    movel([0.091706, -1.408283, -2.552666, -0.751440, 1.570796, 1.662503],accel_mss,speed_ms,0,blend_radius_m)
    movel([0.089171, -1.432149, -2.534440, -0.745800, 1.570796, 1.659968],accel_mss,speed_ms,0,blend_radius_m)
    movel([0.086775, -1.455223, -2.515999, -0.741166, 1.570796, 1.657571],accel_mss,speed_ms,0,blend_radius_m)
    movel([0.116068, -1.448017, -2.521846, -0.742526, 1.570796, 1.686864],accel_mss,speed_ms,0,blend_radius_m)
    movel([0.118372, -1.447476, -2.522281, -0.742631, 1.570796, 1.689168],accel_mss,speed_ms,0,blend_radius_m)
    speed_ms = 0.005
    movel([0.118372, -1.439256, -2.518569, -0.754564, 1.570796, 1.689168],accel_mss,speed_ms,0,blend_radius_m)
    speed_ms = 0.040
    movel([0.108373, -1.430908, -2.525151, -0.756330, 1.570796, 1.679169],accel_mss,speed_ms,0,blend_radius_m)
    speed_ms = 0.005
    movel([0.108373, -1.439191, -2.528898, -0.744300, 1.570796, 1.679169],accel_mss,speed_ms,0,blend_radius_m)
    speed_ms = 0.030
    movel([0.109064, -1.438479, -2.529462, -0.744448, 1.570796, 1.679861],accel_mss,speed_ms,0,blend_radius_m)
    movel([0.109634, -1.437741, -2.530045, -0.744603, 1.570796, 1.680430],accel_mss,speed_ms,0,blend_radius_m)
    movel([0.110059, -1.437005, -2.530627, -0.744758, 1.570796, 1.680855],accel_mss,speed_ms,0,blend_radius_m)
    movel([0.110328, -1.436288, -2.531192, -0.744909, 1.570796, 1.681124],accel_mss,speed_ms,0,blend_radius_m)
    movel([0.110489, -1.435357, -2.531925, -0.745107, 1.570796, 1.681285],accel_mss,speed_ms,0,blend_radius_m)
    movel([0.110459, -1.434480, -2.532614, -0.745295, 1.570796, 1.681255],accel_mss,speed_ms,0,blend_radius_m)
    movel([0.110228, -1.433791, -2.533154, -0.745444, 1.570796, 1.681024],accel_mss,speed_ms,0,blend_radius_m)
    movel([0.109775, -1.433248, -2.533580, -0.745561, 1.570796, 1.680572],accel_mss,speed_ms,0,blend_radius_m)
    movel([0.109099, -1.432863, -2.533881, -0.745645, 1.570796, 1.679896],accel_mss,speed_ms,0,blend_radius_m)
    movel([0.108266, -1.432676, -2.534028, -0.745685, 1.570796, 1.679062],accel_mss,speed_ms,0,blend_radius_m)
    movel([0.107167, -1.432651, -2.534047, -0.745691, 1.570796, 1.677964],accel_mss,speed_ms,0,blend_radius_m)
    movel([0.106011, -1.432776, -2.533950, -0.745663, 1.570796, 1.676807],accel_mss,speed_ms,0,blend_radius_m)
    movel([0.104600, -1.433064, -2.533724, -0.745601, 1.570796, 1.675397],accel_mss,speed_ms,0,blend_radius_m)
    movel([0.103766, -1.433387, -2.533471, -0.745531, 1.570796, 1.674563],accel_mss,speed_ms,0,blend_radius_m)
    movel([0.103005, -1.433924, -2.533050, -0.745415, 1.570796, 1.673801],accel_mss,speed_ms,0,blend_radius_m)
    movel([0.101867, -1.435005, -2.532202, -0.745183, 1.570796, 1.672664],accel_mss,speed_ms,0,blend_radius_m)
    movel([0.100937, -1.436006, -2.531414, -0.744969, 1.570796, 1.671733],accel_mss,speed_ms,0,blend_radius_m)
    movel([0.100376, -1.436776, -2.530807, -0.744806, 1.570796, 1.671172],accel_mss,speed_ms,0,blend_radius_m)
    movel([0.100054, -1.437509, -2.530228, -0.744651, 1.570796, 1.670850],accel_mss,speed_ms,0,blend_radius_m)
    movel([0.099878, -1.438369, -2.529549, -0.744471, 1.570796, 1.670674],accel_mss,speed_ms,0,blend_radius_m)
    movel([0.099866, -1.438969, -2.529074, -0.744346, 1.570796, 1.670663],accel_mss,speed_ms,0,blend_radius_m)
    movel([0.099966, -1.439526, -2.528633, -0.744230, 1.570796, 1.670762],accel_mss,speed_ms,0,blend_radius_m)
    movel([0.100487, -1.440458, -2.527893, -0.744038, 1.570796, 1.671284],accel_mss,speed_ms,0,blend_radius_m)
    movel([0.100905, -1.440826, -2.527601, -0.743962, 1.570796, 1.671701],accel_mss,speed_ms,0,blend_radius_m)
    movel([0.101980, -1.441312, -2.527214, -0.743863, 1.570796, 1.672776],accel_mss,speed_ms,0,blend_radius_m)
    movel([0.102614, -1.441422, -2.527127, -0.743840, 1.570796, 1.673411],accel_mss,speed_ms,0,blend_radius_m)
    movel([0.104044, -1.441369, -2.527169, -0.743851, 1.570796, 1.674840],accel_mss,speed_ms,0,blend_radius_m)
    movel([0.104799, -1.441206, -2.527298, -0.743884, 1.570796, 1.675596],accel_mss,speed_ms,0,blend_radius_m)
    movel([0.106310, -1.440622, -2.527762, -0.744004, 1.570796, 1.677107],accel_mss,speed_ms,0,blend_radius_m)
    movel([0.107038, -1.440213, -2.528087, -0.744088, 1.570796, 1.677835],accel_mss,speed_ms,0,blend_radius_m)
    movel([0.108373, -1.439191, -2.528898, -0.744300, 1.570796, 1.679169],accel_mss,speed_ms,0,blend_radius_m)
    movel([0.109064, -1.438479, -2.529462, -0.744448, 1.570796, 1.679861],accel_mss,speed_ms,0,blend_radius_m)
    movel([0.109634, -1.437741, -2.530045, -0.744603, 1.570796, 1.680430],accel_mss,speed_ms,0,blend_radius_m)
    movel([0.109919, -1.437246, -2.530436, -0.744707, 1.570796, 1.680715],accel_mss,speed_ms,0,blend_radius_m)
    speed_ms = 0.005
    movel([0.109919, -1.428948, -2.526681, -0.756760, 1.570796, 1.680715],accel_mss,speed_ms,0,blend_radius_m)
    speed_ms = 0.040
    movel([0.118670, -1.416855, -2.535995, -0.759539, 1.570796, 1.689466],accel_mss,speed_ms,0,blend_radius_m)
    speed_ms = 0.005
    movel([0.118670, -1.425243, -2.539801, -0.747344, 1.570796, 1.689466],accel_mss,speed_ms,0,blend_radius_m)
    speed_ms = 0.030
    movel([0.124083, -1.423937, -2.540808, -0.747644, 1.570796, 1.694879],accel_mss,speed_ms,0,blend_radius_m)
    movel([0.117797, -1.434992, -2.532211, -0.745185, 1.570796, 1.688593],accel_mss,speed_ms,0,blend_radius_m)
    movel([0.117485, -1.435414, -2.531880, -0.745095, 1.570796, 1.688282],accel_mss,speed_ms,0,blend_radius_m)
    movel([0.116691, -1.434317, -2.532742, -0.745330, 1.570796, 1.687488],accel_mss,speed_ms,0,blend_radius_m)
    movel([0.115225, -1.431178, -2.535198, -0.746013, 1.570796, 1.686021],accel_mss,speed_ms,0,blend_radius_m)
    movel([0.113262, -1.426570, -2.538777, -0.747042, 1.570796, 1.684058],accel_mss,speed_ms,0,blend_radius_m)
    movel([0.118670, -1.425243, -2.539801, -0.747344, 1.570796, 1.689466],accel_mss,speed_ms,0,blend_radius_m)
    movel([0.121038, -1.424669, -2.540244, -0.747476, 1.570796, 1.691834],accel_mss,speed_ms,0,blend_radius_m)
    speed_ms = 0.005
    movel([0.121038, -1.416276, -2.536436, -0.759677, 1.570796, 1.691834],accel_mss,speed_ms,0,blend_radius_m)
    speed_ms = 0.040
    movel([0.111498, -1.424285, -2.530298, -0.757806, 1.570796, 1.682294],accel_mss,speed_ms,0,blend_radius_m)
    speed_ms = 0.005
    movel([0.111498, -1.432618, -2.534073, -0.745698, 1.570796, 1.682294],accel_mss,speed_ms,0,blend_radius_m)
    speed_ms = 0.030
    movel([0.111769, -1.433135, -2.533668, -0.745586, 1.570796, 1.682566],accel_mss,speed_ms,0,blend_radius_m)
    movel([0.112066, -1.434546, -2.532562, -0.745281, 1.570796, 1.682862],accel_mss,speed_ms,0,blend_radius_m)
    movel([0.112043, -1.435207, -2.532042, -0.745139, 1.570796, 1.682839],accel_mss,speed_ms,0,blend_radius_m)
    movel([0.111849, -1.436112, -2.531330, -0.744947, 1.570796, 1.682646],accel_mss,speed_ms,0,blend_radius_m)
    movel([0.111503, -1.437034, -2.530604, -0.744751, 1.570796, 1.682299],accel_mss,speed_ms,0,blend_radius_m)
    movel([0.111013, -1.437950, -2.529880, -0.744559, 1.570796, 1.681809],accel_mss,speed_ms,0,blend_radius_m)
    movel([0.110389, -1.438840, -2.529176, -0.744373, 1.570796, 1.681185],accel_mss,speed_ms,0,blend_radius_m)
    movel([0.109649, -1.439681, -2.528510, -0.744198, 1.570796, 1.680445],accel_mss,speed_ms,0,blend_radius_m)
    movel([0.108810, -1.440452, -2.527898, -0.744039, 1.570796, 1.679607],accel_mss,speed_ms,0,blend_radius_m)
    movel([0.107889, -1.441141, -2.527350, -0.743898, 1.570796, 1.678685],accel_mss,speed_ms,0,blend_radius_m)
    movel([0.106909, -1.441727, -2.526884, -0.743778, 1.570796, 1.677706],accel_mss,speed_ms,0,blend_radius_m)
    movel([0.105881, -1.442207, -2.526502, -0.743680, 1.570796, 1.676677],accel_mss,speed_ms,0,blend_radius_m)
    movel([0.104840, -1.442562, -2.526218, -0.743608, 1.570796, 1.675636],accel_mss,speed_ms,0,blend_radius_m)
    movel([0.103811, -1.442784, -2.526041, -0.743563, 1.570796, 1.674607],accel_mss,speed_ms,0,blend_radius_m)
    movel([0.102814, -1.442870, -2.525973, -0.743546, 1.570796, 1.673610],accel_mss,speed_ms,0,blend_radius_m)
    movel([0.101860, -1.442821, -2.526012, -0.743556, 1.570796, 1.672657],accel_mss,speed_ms,0,blend_radius_m)
    movel([0.100981, -1.442635, -2.526161, -0.743594, 1.570796, 1.671777],accel_mss,speed_ms,0,blend_radius_m)
    movel([0.100198, -1.442319, -2.526412, -0.743658, 1.570796, 1.670994],accel_mss,speed_ms,0,blend_radius_m)
    movel([0.099523, -1.441881, -2.526762, -0.743747, 1.570796, 1.670319],accel_mss,speed_ms,0,blend_radius_m)
    movel([0.098634, -1.440907, -2.527537, -0.743946, 1.570796, 1.669430],accel_mss,speed_ms,0,blend_radius_m)
    movel([0.098355, -1.440381, -2.527954, -0.744054, 1.570796, 1.669152],accel_mss,speed_ms,0,blend_radius_m)
    movel([0.098129, -1.439183, -2.528904, -0.744301, 1.570796, 1.668926],accel_mss,speed_ms,0,blend_radius_m)
    movel([0.098186, -1.438537, -2.529416, -0.744436, 1.570796, 1.668982],accel_mss,speed_ms,0,blend_radius_m)
    movel([0.098626, -1.437145, -2.530516, -0.744728, 1.570796, 1.669422],accel_mss,speed_ms,0,blend_radius_m)
    movel([0.099087, -1.436285, -2.531194, -0.744910, 1.570796, 1.669883],accel_mss,speed_ms,0,blend_radius_m)
    movel([0.099671, -1.435447, -2.531853, -0.745088, 1.570796, 1.670467],accel_mss,speed_ms,0,blend_radius_m)
    movel([0.100365, -1.434653, -2.532478, -0.745258, 1.570796, 1.671161],accel_mss,speed_ms,0,blend_radius_m)
    movel([0.101155, -1.433915, -2.533057, -0.745417, 1.570796, 1.671952],accel_mss,speed_ms,0,blend_radius_m)
    movel([0.102056, -1.433221, -2.533601, -0.745567, 1.570796, 1.672852],accel_mss,speed_ms,0,blend_radius_m)
    movel([0.103011, -1.432609, -2.534081, -0.745700, 1.570796, 1.673808],accel_mss,speed_ms,0,blend_radius_m)
    movel([0.104006, -1.432092, -2.534485, -0.745813, 1.570796, 1.674803],accel_mss,speed_ms,0,blend_radius_m)
    movel([0.105024, -1.431675, -2.534810, -0.745904, 1.570796, 1.675820],accel_mss,speed_ms,0,blend_radius_m)
    movel([0.106037, -1.431373, -2.535046, -0.745970, 1.570796, 1.676834],accel_mss,speed_ms,0,blend_radius_m)
    movel([0.107034, -1.431190, -2.535189, -0.746010, 1.570796, 1.677830],accel_mss,speed_ms,0,blend_radius_m)
    movel([0.108000, -1.431125, -2.535240, -0.746025, 1.570796, 1.678796],accel_mss,speed_ms,0,blend_radius_m)
    movel([0.108911, -1.431181, -2.535196, -0.746012, 1.570796, 1.679707],accel_mss,speed_ms,0,blend_radius_m)
    movel([0.109713, -1.431357, -2.535058, -0.745973, 1.570796, 1.680510],accel_mss,speed_ms,0,blend_radius_m)
    movel([0.110423, -1.431660, -2.534822, -0.745907, 1.570796, 1.681220],accel_mss,speed_ms,0,blend_radius_m)
    movel([0.111022, -1.432085, -2.534490, -0.745814, 1.570796, 1.681818],accel_mss,speed_ms,0,blend_radius_m)
    movel([0.111498, -1.432618, -2.534073, -0.745698, 1.570796, 1.682294],accel_mss,speed_ms,0,blend_radius_m)
    movel([0.111769, -1.433135, -2.533668, -0.745586, 1.570796, 1.682566],accel_mss,speed_ms,0,blend_radius_m)
    movel([0.112020, -1.434323, -2.532737, -0.745329, 1.570796, 1.682816],accel_mss,speed_ms,0,blend_radius_m)
    speed_ms = 0.005
    movel([0.112020, -1.426003, -2.528969, -0.757417, 1.570796, 1.682816],accel_mss,speed_ms,0,blend_radius_m)
    speed_ms = 0.040
    movel([0.108450, -1.426614, -2.528496, -0.757279, 1.570796, 1.679246],accel_mss,speed_ms,0,blend_radius_m)
    speed_ms = 0.005
    movel([0.108450, -1.434929, -2.532261, -0.745199, 1.570796, 1.679246],accel_mss,speed_ms,0,blend_radius_m)
    speed_ms = 0.030
    movel([0.107952, -1.434276, -2.532774, -0.745339, 1.570796, 1.678748],accel_mss,speed_ms,0,blend_radius_m)
    movel([0.107572, -1.434065, -2.532940, -0.745384, 1.570796, 1.678368],accel_mss,speed_ms,0,blend_radius_m)
    movel([0.107121, -1.433941, -2.533037, -0.745411, 1.570796, 1.677918],accel_mss,speed_ms,0,blend_radius_m)
    movel([0.106038, -1.433948, -2.533031, -0.745410, 1.570796, 1.676835],accel_mss,speed_ms,0,blend_radius_m)
    movel([0.104871, -1.434291, -2.532762, -0.745336, 1.570796, 1.675667],accel_mss,speed_ms,0,blend_radius_m)
    movel([0.103728, -1.434938, -2.532254, -0.745197, 1.570796, 1.674524],accel_mss,speed_ms,0,blend_radius_m)
    movel([0.102745, -1.435815, -2.531564, -0.745010, 1.570796, 1.673541],accel_mss,speed_ms,0,blend_radius_m)
    movel([0.102363, -1.436294, -2.531187, -0.744908, 1.570796, 1.673159],accel_mss,speed_ms,0,blend_radius_m)
    movel([0.101858, -1.437301, -2.530393, -0.744695, 1.570796, 1.672655],accel_mss,speed_ms,0,blend_radius_m)
    movel([0.101749, -1.437800, -2.529999, -0.744590, 1.570796, 1.672545],accel_mss,speed_ms,0,blend_radius_m)
    movel([0.101790, -1.438633, -2.529340, -0.744416, 1.570796, 1.672586],accel_mss,speed_ms,0,blend_radius_m)
    movel([0.102119, -1.439326, -2.528791, -0.744272, 1.570796, 1.672915],accel_mss,speed_ms,0,blend_radius_m)
    movel([0.102703, -1.439804, -2.528412, -0.744173, 1.570796, 1.673500],accel_mss,speed_ms,0,blend_radius_m)
    movel([0.103505, -1.440030, -2.528233, -0.744126, 1.570796, 1.674302],accel_mss,speed_ms,0,blend_radius_m)
    movel([0.104454, -1.439989, -2.528265, -0.744135, 1.570796, 1.675251],accel_mss,speed_ms,0,blend_radius_m)
    movel([0.105461, -1.439681, -2.528509, -0.744198, 1.570796, 1.676258],accel_mss,speed_ms,0,blend_radius_m)
    movel([0.106463, -1.439130, -2.528947, -0.744313, 1.570796, 1.677259],accel_mss,speed_ms,0,blend_radius_m)
    movel([0.107355, -1.438395, -2.529529, -0.744466, 1.570796, 1.678151],accel_mss,speed_ms,0,blend_radius_m)
    movel([0.108163, -1.437463, -2.530265, -0.744661, 1.570796, 1.678959],accel_mss,speed_ms,0,blend_radius_m)
    movel([0.108589, -1.436654, -2.530904, -0.744832, 1.570796, 1.679385],accel_mss,speed_ms,0,blend_radius_m)
    movel([0.108678, -1.435849, -2.531537, -0.745002, 1.570796, 1.679474],accel_mss,speed_ms,0,blend_radius_m)
    movel([0.108450, -1.434929, -2.532261, -0.745199, 1.570796, 1.679246],accel_mss,speed_ms,0,blend_radius_m)
    movel([0.107952, -1.434276, -2.532774, -0.745339, 1.570796, 1.678748],accel_mss,speed_ms,0,blend_radius_m)
    movel([0.107572, -1.434065, -2.532940, -0.745384, 1.570796, 1.678368],accel_mss,speed_ms,0,blend_radius_m)
    movel([0.107121, -1.433941, -2.533037, -0.745411, 1.570796, 1.677918],accel_mss,speed_ms,0,blend_radius_m)
    speed_ms = 0.005
    movel([0.107012, -1.425618, -2.529268, -0.757504, 1.570796, 1.677809],accel_mss,speed_ms,0,blend_radius_m)
    speed_ms = 0.040
    movel([0.083343, -1.436462, -2.520784, -0.755143, 1.570796, 1.654139],accel_mss,speed_ms,0,blend_radius_m)
    speed_ms = 0.005
    movel([0.083343, -1.444703, -2.524508, -0.743178, 1.570796, 1.654139],accel_mss,speed_ms,0,blend_radius_m)
    speed_ms = 0.030
    movel([0.085200, -1.444214, -2.524899, -0.743276, 1.570796, 1.655996],accel_mss,speed_ms,0,blend_radius_m)
    movel([0.085840, -1.437885, -2.529932, -0.744572, 1.570796, 1.656636],accel_mss,speed_ms,0,blend_radius_m)
    movel([0.086489, -1.431498, -2.534949, -0.745943, 1.570796, 1.657285],accel_mss,speed_ms,0,blend_radius_m)
    movel([0.084603, -1.432003, -2.534554, -0.745832, 1.570796, 1.655399],accel_mss,speed_ms,0,blend_radius_m)
    movel([0.082718, -1.432510, -2.534157, -0.745721, 1.570796, 1.653514],accel_mss,speed_ms,0,blend_radius_m)
    movel([0.082098, -1.438881, -2.529144, -0.744364, 1.570796, 1.652894],accel_mss,speed_ms,0,blend_radius_m)
    movel([0.081487, -1.445194, -2.524114, -0.743080, 1.570796, 1.652283],accel_mss,speed_ms,0,blend_radius_m)
    movel([0.083343, -1.444703, -2.524508, -0.743178, 1.570796, 1.654139],accel_mss,speed_ms,0,blend_radius_m)
    movel([0.085200, -1.444214, -2.524899, -0.743276, 1.570796, 1.655996],accel_mss,speed_ms,0,blend_radius_m)
    movel([0.085240, -1.443820, -2.525214, -0.743355, 1.570796, 1.656036],accel_mss,speed_ms,0,blend_radius_m)
    speed_ms = 0.005
    movel([0.085240, -1.435572, -2.521486, -0.755330, 1.570796, 1.656036],accel_mss,speed_ms,0,blend_radius_m)
    speed_ms = 0.040
    movel([0.080369, -1.396684, -2.551051, -0.764654, 1.570796, 1.651165],accel_mss,speed_ms,0,blend_radius_m)
    speed_ms = 0.005
    movel([0.080369, -1.405221, -2.554943, -0.752225, 1.570796, 1.651165],accel_mss,speed_ms,0,blend_radius_m)
    speed_ms = 0.030
    movel([0.082668, -1.404286, -2.555636, -0.752468, 1.570796, 1.653464],accel_mss,speed_ms,0,blend_radius_m)
    movel([0.083132, -1.399509, -2.559154, -0.753727, 1.570796, 1.653929],accel_mss,speed_ms,0,blend_radius_m)
    movel([0.083285, -1.397676, -2.560495, -0.754219, 1.570796, 1.654081],accel_mss,speed_ms,0,blend_radius_m)
    movel([0.083369, -1.394878, -2.562532, -0.754979, 1.570796, 1.654165],accel_mss,speed_ms,0,blend_radius_m)
    movel([0.071293, -1.397205, -2.560838, -0.754346, 1.570796, 1.642090],accel_mss,speed_ms,0,blend_radius_m)
    movel([0.066805, -1.398147, -2.560151, -0.754092, 1.570796, 1.637601],accel_mss,speed_ms,0,blend_radius_m)
    movel([0.059543, -1.399830, -2.558918, -0.753641, 1.570796, 1.630340],accel_mss,speed_ms,0,blend_radius_m)
    movel([0.058947, -1.400083, -2.558732, -0.753573, 1.570796, 1.629743],accel_mss,speed_ms,0,blend_radius_m)
    movel([0.058527, -1.400449, -2.558464, -0.753476, 1.570796, 1.629324],accel_mss,speed_ms,0,blend_radius_m)
    movel([0.058288, -1.400892, -2.558139, -0.753359, 1.570796, 1.629084],accel_mss,speed_ms,0,blend_radius_m)
    movel([0.058040, -1.402395, -2.557032, -0.752962, 1.570796, 1.628837],accel_mss,speed_ms,0,blend_radius_m)
    movel([0.058173, -1.404016, -2.555835, -0.752538, 1.570796, 1.628969],accel_mss,speed_ms,0,blend_radius_m)
    movel([0.058390, -1.404688, -2.555338, -0.752363, 1.570796, 1.629186],accel_mss,speed_ms,0,blend_radius_m)
    movel([0.058721, -1.405288, -2.554893, -0.752208, 1.570796, 1.629517],accel_mss,speed_ms,0,blend_radius_m)
    movel([0.059262, -1.405908, -2.554434, -0.752048, 1.570796, 1.630058],accel_mss,speed_ms,0,blend_radius_m)
    movel([0.059943, -1.406402, -2.554066, -0.751921, 1.570796, 1.630739],accel_mss,speed_ms,0,blend_radius_m)
    movel([0.060908, -1.406890, -2.553704, -0.751796, 1.570796, 1.631705],accel_mss,speed_ms,0,blend_radius_m)
    movel([0.061951, -1.407284, -2.553410, -0.751695, 1.570796, 1.632747],accel_mss,speed_ms,0,blend_radius_m)
    movel([0.064429, -1.407851, -2.552988, -0.751550, 1.570796, 1.635225],accel_mss,speed_ms,0,blend_radius_m)
    movel([0.065734, -1.407984, -2.552889, -0.751516, 1.570796, 1.636530],accel_mss,speed_ms,0,blend_radius_m)
    movel([0.068559, -1.407941, -2.552921, -0.751527, 1.570796, 1.639356],accel_mss,speed_ms,0,blend_radius_m)
    movel([0.070060, -1.407772, -2.553047, -0.751570, 1.570796, 1.640856],accel_mss,speed_ms,0,blend_radius_m)
    movel([0.073745, -1.407121, -2.553532, -0.751736, 1.570796, 1.644541],accel_mss,speed_ms,0,blend_radius_m)
    movel([0.077424, -1.406227, -2.554196, -0.751965, 1.570796, 1.648221],accel_mss,speed_ms,0,blend_radius_m)
    movel([0.080369, -1.405221, -2.554943, -0.752225, 1.570796, 1.651165],accel_mss,speed_ms,0,blend_radius_m)
    movel([0.082668, -1.404286, -2.555636, -0.752468, 1.570796, 1.653464],accel_mss,speed_ms,0,blend_radius_m)
    speed_ms = 0.005
    movel([0.082679, -1.395622, -2.551827, -0.764940, 1.570796, 1.653475],accel_mss,speed_ms,0,blend_radius_m)
    speed_ms = 0.040
    movel([0.064626, -1.389214, -2.556477, -0.766699, 1.570796, 1.635422],accel_mss,speed_ms,0,blend_radius_m)
    speed_ms = 0.005
    movel([0.064626, -1.397805, -2.560400, -0.754184, 1.570796, 1.635422],accel_mss,speed_ms,0,blend_radius_m)
    speed_ms = 0.030
    movel([0.068867, -1.396843, -2.561102, -0.754444, 1.570796, 1.639663],accel_mss,speed_ms,0,blend_radius_m)
    movel([0.070556, -1.396424, -2.561408, -0.754557, 1.570796, 1.641353],accel_mss,speed_ms,0,blend_radius_m)
    movel([0.069209, -1.396473, -2.561372, -0.754544, 1.570796, 1.640005],accel_mss,speed_ms,0,blend_radius_m)
    movel([0.067359, -1.396817, -2.561121, -0.754451, 1.570796, 1.638155],accel_mss,speed_ms,0,blend_radius_m)
    movel([0.060872, -1.398254, -2.560073, -0.754063, 1.570796, 1.631668],accel_mss,speed_ms,0,blend_radius_m)
    movel([0.059184, -1.398684, -2.559758, -0.753947, 1.570796, 1.629980],accel_mss,speed_ms,0,blend_radius_m)
    movel([0.064626, -1.397805, -2.560400, -0.754184, 1.570796, 1.635422],accel_mss,speed_ms,0,blend_radius_m)
    movel([0.067065, -1.397250, -2.560805, -0.754333, 1.570796, 1.637861],accel_mss,speed_ms,0,blend_radius_m)
    speed_ms = 0.005
    movel([0.067065, -1.388655, -2.556879, -0.766855, 1.570796, 1.637861],accel_mss,speed_ms,0,blend_radius_m)
    speed_ms = 0.040
    movel([0.077329, -1.386656, -2.558316, -0.767417, 1.570796, 1.648125],accel_mss,speed_ms,0,blend_radius_m)
    speed_ms = 0.005
    movel([0.077329, -1.395266, -2.562250, -0.754873, 1.570796, 1.648125],accel_mss,speed_ms,0,blend_radius_m)
    speed_ms = 0.030
    movel([0.081574, -1.394344, -2.562920, -0.755125, 1.570796, 1.652370],accel_mss,speed_ms,0,blend_radius_m)
    movel([0.083266, -1.393940, -2.563212, -0.755236, 1.570796, 1.654062],accel_mss,speed_ms,0,blend_radius_m)
    movel([0.081921, -1.393974, -2.563188, -0.755227, 1.570796, 1.652718],accel_mss,speed_ms,0,blend_radius_m)
    movel([0.080071, -1.394300, -2.562951, -0.755137, 1.570796, 1.650867],accel_mss,speed_ms,0,blend_radius_m)
    movel([0.073577, -1.395676, -2.561952, -0.754761, 1.570796, 1.644374],accel_mss,speed_ms,0,blend_radius_m)
    movel([0.071887, -1.396091, -2.561650, -0.754648, 1.570796, 1.642683],accel_mss,speed_ms,0,blend_radius_m)
    movel([0.077329, -1.395266, -2.562250, -0.754873, 1.570796, 1.648125],accel_mss,speed_ms,0,blend_radius_m)
    movel([0.079771, -1.394734, -2.562637, -0.755018, 1.570796, 1.650567],accel_mss,speed_ms,0,blend_radius_m)
    speed_ms = 0.005
    movel([0.079771, -1.386121, -2.558700, -0.767569, 1.570796, 1.650567],accel_mss,speed_ms,0,blend_radius_m)
    speed_ms = 0.040
    movel([0.082596, -1.384305, -2.559998, -0.768086, 1.570796, 1.653392],accel_mss,speed_ms,0,blend_radius_m)
    speed_ms = 0.005
    movel([0.082596, -1.392931, -2.563943, -0.755515, 1.570796, 1.653392],accel_mss,speed_ms,0,blend_radius_m)
    speed_ms = 0.030
    movel([0.080067, -1.393544, -2.563500, -0.755346, 1.570796, 1.650864],accel_mss,speed_ms,0,blend_radius_m)
    movel([0.070347, -1.395469, -2.562102, -0.754817, 1.570796, 1.641143],accel_mss,speed_ms,0,blend_radius_m)
    movel([0.059849, -1.397609, -2.560544, -0.754237, 1.570796, 1.630646],accel_mss,speed_ms,0,blend_radius_m)
    movel([0.059405, -1.397561, -2.560579, -0.754250, 1.570796, 1.630201],accel_mss,speed_ms,0,blend_radius_m)
    movel([0.059560, -1.397205, -2.560838, -0.754346, 1.570796, 1.630356],accel_mss,speed_ms,0,blend_radius_m)
    movel([0.061171, -1.396673, -2.561226, -0.754490, 1.570796, 1.631968],accel_mss,speed_ms,0,blend_radius_m)
    movel([0.064490, -1.395852, -2.561824, -0.754713, 1.570796, 1.635287],accel_mss,speed_ms,0,blend_radius_m)
    movel([0.083770, -1.391761, -2.564789, -0.755840, 1.570796, 1.654566],accel_mss,speed_ms,0,blend_radius_m)
    movel([0.083851, -1.392158, -2.564502, -0.755729, 1.570796, 1.654647],accel_mss,speed_ms,0,blend_radius_m)
    movel([0.083064, -1.392765, -2.564063, -0.755561, 1.570796, 1.653860],accel_mss,speed_ms,0,blend_radius_m)
    movel([0.082596, -1.392931, -2.563943, -0.755515, 1.570796, 1.653392],accel_mss,speed_ms,0,blend_radius_m)
    movel([0.080141, -1.393526, -2.563512, -0.755350, 1.570796, 1.650937],accel_mss,speed_ms,0,blend_radius_m)
    speed_ms = 0.005
    movel([0.080141, -1.384904, -2.559570, -0.767915, 1.570796, 1.650937],accel_mss,speed_ms,0,blend_radius_m)
    speed_ms = 0.040
    movel([0.080979, -1.381872, -2.561731, -0.768786, 1.570796, 1.651775],accel_mss,speed_ms,0,blend_radius_m)
    speed_ms = 0.005
    movel([0.080979, -1.390515, -2.565686, -0.756187, 1.570796, 1.651775],accel_mss,speed_ms,0,blend_radius_m)
    speed_ms = 0.030
    movel([0.082613, -1.390041, -2.566028, -0.756321, 1.570796, 1.653409],accel_mss,speed_ms,0,blend_radius_m)
    movel([0.084226, -1.373470, -2.577746, -0.761173, 1.570796, 1.655023],accel_mss,speed_ms,0,blend_radius_m)
    movel([0.085905, -1.356480, -2.589353, -0.766556, 1.570796, 1.656701],accel_mss,speed_ms,0,blend_radius_m)
    movel([0.073910, -1.360292, -2.586784, -0.765313, 1.570796, 1.644706],accel_mss,speed_ms,0,blend_radius_m)
    movel([0.061960, -1.364186, -2.584139, -0.764064, 1.570796, 1.632757],accel_mss,speed_ms,0,blend_radius_m)
    movel([0.060698, -1.379920, -2.573232, -0.759238, 1.570796, 1.631494],accel_mss,speed_ms,0,blend_radius_m)
    movel([0.060254, -1.385848, -2.569030, -0.757511, 1.570796, 1.631050],accel_mss,speed_ms,0,blend_radius_m)
    movel([0.059726, -1.395090, -2.562378, -0.754921, 1.570796, 1.630522],accel_mss,speed_ms,0,blend_radius_m)
    movel([0.073579, -1.392180, -2.564486, -0.755723, 1.570796, 1.644375],accel_mss,speed_ms,0,blend_radius_m)
    movel([0.077024, -1.391431, -2.565027, -0.755932, 1.570796, 1.647820],accel_mss,speed_ms,0,blend_radius_m)
    movel([0.080979, -1.390515, -2.565686, -0.756187, 1.570796, 1.651775],accel_mss,speed_ms,0,blend_radius_m)
    movel([0.082613, -1.390041, -2.566028, -0.756321, 1.570796, 1.653409],accel_mss,speed_ms,0,blend_radius_m)
    movel([0.082683, -1.389316, -2.566549, -0.756525, 1.570796, 1.653479],accel_mss,speed_ms,0,blend_radius_m)
    speed_ms = 0.005
    movel([0.082683, -1.380664, -2.562588, -0.769137, 1.570796, 1.653479],accel_mss,speed_ms,0,blend_radius_m)
    speed_ms = 0.040
    movel([0.104255, -1.354850, -2.580410, -0.777129, 1.570796, 1.675051],accel_mss,speed_ms,0,blend_radius_m)
    speed_ms = 0.005
    movel([0.104255, -1.363681, -2.584483, -0.764225, 1.570796, 1.675051],accel_mss,speed_ms,0,blend_radius_m)
    speed_ms = 0.030
    movel([0.104837, -1.364381, -2.584006, -0.764002, 1.570796, 1.675633],accel_mss,speed_ms,0,blend_radius_m)
    movel([0.105164, -1.365257, -2.583408, -0.763724, 1.570796, 1.675960],accel_mss,speed_ms,0,blend_radius_m)
    movel([0.105210, -1.366242, -2.582733, -0.763413, 1.570796, 1.676006],accel_mss,speed_ms,0,blend_radius_m)
    movel([0.104969, -1.367313, -2.581999, -0.763077, 1.570796, 1.675765],accel_mss,speed_ms,0,blend_radius_m)
    movel([0.104455, -1.368422, -2.581237, -0.762730, 1.570796, 1.675251],accel_mss,speed_ms,0,blend_radius_m)
    movel([0.103698, -1.369493, -2.580500, -0.762397, 1.570796, 1.674494],accel_mss,speed_ms,0,blend_radius_m)
    movel([0.102710, -1.370523, -2.579788, -0.762078, 1.570796, 1.673506],accel_mss,speed_ms,0,blend_radius_m)
    movel([0.101583, -1.371423, -2.579166, -0.761800, 1.570796, 1.672379],accel_mss,speed_ms,0,blend_radius_m)
    movel([0.100743, -1.372075, -2.578714, -0.761600, 1.570796, 1.671539],accel_mss,speed_ms,0,blend_radius_m)
    movel([0.100262, -1.372631, -2.578328, -0.761430, 1.570796, 1.671058],accel_mss,speed_ms,0,blend_radius_m)
    movel([0.099987, -1.373275, -2.577881, -0.761233, 1.570796, 1.670783],accel_mss,speed_ms,0,blend_radius_m)
    movel([0.099815, -1.374253, -2.577201, -0.760935, 1.570796, 1.670612],accel_mss,speed_ms,0,blend_radius_m)
    movel([0.099670, -1.375197, -2.576543, -0.760649, 1.570796, 1.670466],accel_mss,speed_ms,0,blend_radius_m)
    movel([0.099463, -1.375717, -2.576180, -0.760492, 1.570796, 1.670260],accel_mss,speed_ms,0,blend_radius_m)
    movel([0.099131, -1.376043, -2.575952, -0.760394, 1.570796, 1.669927],accel_mss,speed_ms,0,blend_radius_m)
    movel([0.098607, -1.376274, -2.575790, -0.760324, 1.570796, 1.669404],accel_mss,speed_ms,0,blend_radius_m)
    movel([0.098103, -1.376335, -2.575748, -0.760306, 1.570796, 1.668900],accel_mss,speed_ms,0,blend_radius_m)
    movel([0.097826, -1.376177, -2.575858, -0.760354, 1.570796, 1.668623],accel_mss,speed_ms,0,blend_radius_m)
    movel([0.097730, -1.375738, -2.576165, -0.760486, 1.570796, 1.668526],accel_mss,speed_ms,0,blend_radius_m)
    movel([0.097799, -1.374804, -2.576817, -0.760768, 1.570796, 1.668595],accel_mss,speed_ms,0,blend_radius_m)
    movel([0.097855, -1.373879, -2.577461, -0.761049, 1.570796, 1.668651],accel_mss,speed_ms,0,blend_radius_m)
    movel([0.097739, -1.373373, -2.577813, -0.761203, 1.570796, 1.668535],accel_mss,speed_ms,0,blend_radius_m)
    movel([0.097424, -1.373105, -2.577999, -0.761285, 1.570796, 1.668221],accel_mss,speed_ms,0,blend_radius_m)
    movel([0.095809, -1.372801, -2.578210, -0.761378, 1.570796, 1.666605],accel_mss,speed_ms,0,blend_radius_m)
    movel([0.094976, -1.372335, -2.578533, -0.761520, 1.570796, 1.665772],accel_mss,speed_ms,0,blend_radius_m)
    movel([0.094371, -1.371609, -2.579037, -0.761743, 1.570796, 1.665168],accel_mss,speed_ms,0,blend_radius_m)
    movel([0.094042, -1.370689, -2.579673, -0.762026, 1.570796, 1.664839],accel_mss,speed_ms,0,blend_radius_m)
    movel([0.094002, -1.369617, -2.580414, -0.762358, 1.570796, 1.664798],accel_mss,speed_ms,0,blend_radius_m)
    movel([0.094259, -1.368453, -2.581215, -0.762720, 1.570796, 1.665056],accel_mss,speed_ms,0,blend_radius_m)
    movel([0.094796, -1.367284, -2.582019, -0.763086, 1.570796, 1.665593],accel_mss,speed_ms,0,blend_radius_m)
    movel([0.095599, -1.366150, -2.582796, -0.763442, 1.570796, 1.666396],accel_mss,speed_ms,0,blend_radius_m)
    movel([0.096227, -1.365452, -2.583274, -0.763663, 1.570796, 1.667024],accel_mss,speed_ms,0,blend_radius_m)
    movel([0.096923, -1.364774, -2.583737, -0.763877, 1.570796, 1.667719],accel_mss,speed_ms,0,blend_radius_m)
    movel([0.098078, -1.363868, -2.584356, -0.764165, 1.570796, 1.668874],accel_mss,speed_ms,0,blend_radius_m)
    movel([0.098585, -1.363500, -2.584606, -0.764282, 1.570796, 1.669381],accel_mss,speed_ms,0,blend_radius_m)
    movel([0.098932, -1.363054, -2.584910, -0.764425, 1.570796, 1.669729],accel_mss,speed_ms,0,blend_radius_m)
    movel([0.099160, -1.362448, -2.585322, -0.764619, 1.570796, 1.669956],accel_mss,speed_ms,0,blend_radius_m)
    movel([0.099310, -1.361555, -2.585929, -0.764905, 1.570796, 1.670106],accel_mss,speed_ms,0,blend_radius_m)
    movel([0.099443, -1.360719, -2.586495, -0.765175, 1.570796, 1.670239],accel_mss,speed_ms,0,blend_radius_m)
    movel([0.099642, -1.360152, -2.586879, -0.765358, 1.570796, 1.670438],accel_mss,speed_ms,0,blend_radius_m)
    movel([0.099917, -1.359787, -2.587126, -0.765476, 1.570796, 1.670713],accel_mss,speed_ms,0,blend_radius_m)
    movel([0.100282, -1.359575, -2.587269, -0.765545, 1.570796, 1.671078],accel_mss,speed_ms,0,blend_radius_m)
    movel([0.100621, -1.359585, -2.587262, -0.765542, 1.570796, 1.671417],accel_mss,speed_ms,0,blend_radius_m)
    movel([0.100827, -1.359812, -2.587109, -0.765468, 1.570796, 1.671624],accel_mss,speed_ms,0,blend_radius_m)
    movel([0.100904, -1.360303, -2.586777, -0.765309, 1.570796, 1.671701],accel_mss,speed_ms,0,blend_radius_m)
    movel([0.100845, -1.361129, -2.586217, -0.765042, 1.570796, 1.671642],accel_mss,speed_ms,0,blend_radius_m)
    movel([0.100780, -1.362096, -2.585562, -0.764732, 1.570796, 1.671576],accel_mss,speed_ms,0,blend_radius_m)
    movel([0.100898, -1.362572, -2.585238, -0.764579, 1.570796, 1.671694],accel_mss,speed_ms,0,blend_radius_m)
    movel([0.101234, -1.362784, -2.585094, -0.764511, 1.570796, 1.672030],accel_mss,speed_ms,0,blend_radius_m)
    movel([0.102445, -1.362847, -2.585051, -0.764491, 1.570796, 1.673242],accel_mss,speed_ms,0,blend_radius_m)
    movel([0.103098, -1.363031, -2.584926, -0.764432, 1.570796, 1.673894],accel_mss,speed_ms,0,blend_radius_m)
    movel([0.104255, -1.363681, -2.584483, -0.764225, 1.570796, 1.675051],accel_mss,speed_ms,0,blend_radius_m)
    movel([0.104837, -1.364381, -2.584006, -0.764002, 1.570796, 1.675633],accel_mss,speed_ms,0,blend_radius_m)
    movel([0.105164, -1.365257, -2.583408, -0.763724, 1.570796, 1.675960],accel_mss,speed_ms,0,blend_radius_m)
    speed_ms = 0.005
    movel([0.105164, -1.356437, -2.579342, -0.776611, 1.570796, 1.675960],accel_mss,speed_ms,0,blend_radius_m)
    speed_ms = 0.040
    movel([0.122669, -1.349661, -2.583881, -0.778848, 1.570796, 1.693465],accel_mss,speed_ms,0,blend_radius_m)
    speed_ms = 0.005
    movel([0.122669, -1.358527, -2.587977, -0.765886, 1.570796, 1.693465],accel_mss,speed_ms,0,blend_radius_m)
    speed_ms = 0.030
    movel([0.121598, -1.357814, -2.588456, -0.766118, 1.570796, 1.692395],accel_mss,speed_ms,0,blend_radius_m)
    movel([0.121035, -1.357584, -2.588611, -0.766193, 1.570796, 1.691831],accel_mss,speed_ms,0,blend_radius_m)
    movel([0.120136, -1.357414, -2.588726, -0.766249, 1.570796, 1.690932],accel_mss,speed_ms,0,blend_radius_m)
    movel([0.119877, -1.357136, -2.588913, -0.766340, 1.570796, 1.690674],accel_mss,speed_ms,0,blend_radius_m)
    movel([0.119791, -1.356614, -2.589263, -0.766512, 1.570796, 1.690587],accel_mss,speed_ms,0,blend_radius_m)
    movel([0.119864, -1.355735, -2.589853, -0.766801, 1.570796, 1.690660],accel_mss,speed_ms,0,blend_radius_m)
    movel([0.119956, -1.354790, -2.590486, -0.767113, 1.570796, 1.690753],accel_mss,speed_ms,0,blend_radius_m)
    movel([0.119869, -1.354341, -2.590786, -0.767262, 1.570796, 1.690665],accel_mss,speed_ms,0,blend_radius_m)
    movel([0.119591, -1.354181, -2.590893, -0.767315, 1.570796, 1.690387],accel_mss,speed_ms,0,blend_radius_m)
    movel([0.119076, -1.354238, -2.590855, -0.767296, 1.570796, 1.689873],accel_mss,speed_ms,0,blend_radius_m)
    movel([0.118538, -1.354473, -2.590698, -0.767218, 1.570796, 1.689334],accel_mss,speed_ms,0,blend_radius_m)
    movel([0.118192, -1.354813, -2.590470, -0.767106, 1.570796, 1.688988],accel_mss,speed_ms,0,blend_radius_m)
    movel([0.117970, -1.355356, -2.590107, -0.766926, 1.570796, 1.688766],accel_mss,speed_ms,0,blend_radius_m)
    movel([0.117799, -1.356345, -2.589444, -0.766600, 1.570796, 1.688595],accel_mss,speed_ms,0,blend_radius_m)
    movel([0.117619, -1.357314, -2.588793, -0.766282, 1.570796, 1.688415],accel_mss,speed_ms,0,blend_radius_m)
    movel([0.117363, -1.357943, -2.588370, -0.766076, 1.570796, 1.688160],accel_mss,speed_ms,0,blend_radius_m)
    movel([0.116965, -1.358421, -2.588047, -0.765920, 1.570796, 1.687762],accel_mss,speed_ms,0,blend_radius_m)
    movel([0.116347, -1.358868, -2.587746, -0.765775, 1.570796, 1.687143],accel_mss,speed_ms,0,blend_radius_m)
    movel([0.114910, -1.359918, -2.587037, -0.765434, 1.570796, 1.685707],accel_mss,speed_ms,0,blend_radius_m)
    movel([0.114280, -1.360543, -2.586614, -0.765232, 1.570796, 1.685076],accel_mss,speed_ms,0,blend_radius_m)
    movel([0.113263, -1.361927, -2.585677, -0.764786, 1.570796, 1.684059],accel_mss,speed_ms,0,blend_radius_m)
    movel([0.112890, -1.362657, -2.585180, -0.764552, 1.570796, 1.683686],accel_mss,speed_ms,0,blend_radius_m)
    movel([0.112469, -1.364095, -2.584201, -0.764093, 1.570796, 1.683266],accel_mss,speed_ms,0,blend_radius_m)
    movel([0.112427, -1.364785, -2.583730, -0.763874, 1.570796, 1.683223],accel_mss,speed_ms,0,blend_radius_m)
    movel([0.112679, -1.366026, -2.582882, -0.763481, 1.570796, 1.683475],accel_mss,speed_ms,0,blend_radius_m)
    movel([0.112969, -1.366550, -2.582523, -0.763316, 1.570796, 1.683766],accel_mss,speed_ms,0,blend_radius_m)
    movel([0.113847, -1.367339, -2.581981, -0.763068, 1.570796, 1.684643],accel_mss,speed_ms,0,blend_radius_m)
    movel([0.114418, -1.367593, -2.581807, -0.762989, 1.570796, 1.685215],accel_mss,speed_ms,0,blend_radius_m)
    movel([0.115974, -1.367950, -2.581562, -0.762877, 1.570796, 1.686771],accel_mss,speed_ms,0,blend_radius_m)
    movel([0.116405, -1.368242, -2.581361, -0.762786, 1.570796, 1.687201],accel_mss,speed_ms,0,blend_radius_m)
    movel([0.116560, -1.368747, -2.581013, -0.762629, 1.570796, 1.687356],accel_mss,speed_ms,0,blend_radius_m)
    movel([0.116497, -1.369690, -2.580363, -0.762335, 1.570796, 1.687293],accel_mss,speed_ms,0,blend_radius_m)
    movel([0.116432, -1.370469, -2.579826, -0.762094, 1.570796, 1.687228],accel_mss,speed_ms,0,blend_radius_m)
    movel([0.116500, -1.370938, -2.579501, -0.761950, 1.570796, 1.687297],accel_mss,speed_ms,0,blend_radius_m)
    movel([0.116700, -1.371159, -2.579349, -0.761882, 1.570796, 1.687496],accel_mss,speed_ms,0,blend_radius_m)
    movel([0.117030, -1.371172, -2.579340, -0.761878, 1.570796, 1.687826],accel_mss,speed_ms,0,blend_radius_m)
    movel([0.117391, -1.370967, -2.579481, -0.761941, 1.570796, 1.688187],accel_mss,speed_ms,0,blend_radius_m)
    movel([0.117669, -1.370607, -2.579730, -0.762052, 1.570796, 1.688465],accel_mss,speed_ms,0,blend_radius_m)
    movel([0.117877, -1.370039, -2.580122, -0.762227, 1.570796, 1.688674],accel_mss,speed_ms,0,blend_radius_m)
    movel([0.118030, -1.369185, -2.580712, -0.762492, 1.570796, 1.688826],accel_mss,speed_ms,0,blend_radius_m)
    movel([0.118210, -1.368218, -2.581377, -0.762794, 1.570796, 1.689006],accel_mss,speed_ms,0,blend_radius_m)
    movel([0.118467, -1.367603, -2.581800, -0.762986, 1.570796, 1.689263],accel_mss,speed_ms,0,blend_radius_m)
    movel([0.118876, -1.367130, -2.582125, -0.763134, 1.570796, 1.689673],accel_mss,speed_ms,0,blend_radius_m)
    movel([0.119531, -1.366672, -2.582439, -0.763278, 1.570796, 1.690327],accel_mss,speed_ms,0,blend_radius_m)
    movel([0.120700, -1.365861, -2.582995, -0.763533, 1.570796, 1.691497],accel_mss,speed_ms,0,blend_radius_m)
    movel([0.121723, -1.364870, -2.583672, -0.763847, 1.570796, 1.692519],accel_mss,speed_ms,0,blend_radius_m)
    movel([0.122566, -1.363729, -2.584451, -0.764210, 1.570796, 1.693363],accel_mss,speed_ms,0,blend_radius_m)
    movel([0.123164, -1.362538, -2.585261, -0.764590, 1.570796, 1.693960],accel_mss,speed_ms,0,blend_radius_m)
    movel([0.123489, -1.361349, -2.586068, -0.764971, 1.570796, 1.694285],accel_mss,speed_ms,0,blend_radius_m)
    movel([0.123515, -1.360238, -2.586821, -0.765330, 1.570796, 1.694312],accel_mss,speed_ms,0,blend_radius_m)
    movel([0.123241, -1.359284, -2.587466, -0.765639, 1.570796, 1.694037],accel_mss,speed_ms,0,blend_radius_m)
    movel([0.122669, -1.358527, -2.587977, -0.765886, 1.570796, 1.693465],accel_mss,speed_ms,0,blend_radius_m)
    movel([0.121598, -1.357814, -2.588456, -0.766118, 1.570796, 1.692395],accel_mss,speed_ms,0,blend_radius_m)
    movel([0.121035, -1.357584, -2.588611, -0.766193, 1.570796, 1.691831],accel_mss,speed_ms,0,blend_radius_m)
    speed_ms = 0.005
    movel([0.121035, -1.348712, -2.584511, -0.779166, 1.570796, 1.691831],accel_mss,speed_ms,0,blend_radius_m)
    speed_ms = 0.040
    movel([0.114436, -1.335439, -2.593203, -0.783747, 1.570796, 1.685232],accel_mss,speed_ms,0,blend_radius_m)
    speed_ms = 0.005
    movel([0.114436, -1.344399, -2.597361, -0.770629, 1.570796, 1.685232],accel_mss,speed_ms,0,blend_radius_m)
    speed_ms = 0.030
    movel([0.113833, -1.345365, -2.596728, -0.770296, 1.570796, 1.684629],accel_mss,speed_ms,0,blend_radius_m)
    movel([0.113126, -1.346300, -2.596115, -0.769975, 1.570796, 1.683923],accel_mss,speed_ms,0,blend_radius_m)
    movel([0.111407, -1.348105, -2.594926, -0.769358, 1.570796, 1.682203],accel_mss,speed_ms,0,blend_radius_m)
    movel([0.110416, -1.348947, -2.594370, -0.769072, 1.570796, 1.681212],accel_mss,speed_ms,0,blend_radius_m)
    movel([0.108276, -1.350421, -2.593395, -0.768573, 1.570796, 1.679072],accel_mss,speed_ms,0,blend_radius_m)
    movel([0.107148, -1.351042, -2.592983, -0.768364, 1.570796, 1.677945],accel_mss,speed_ms,0,blend_radius_m)
    movel([0.104917, -1.351966, -2.592369, -0.768054, 1.570796, 1.675714],accel_mss,speed_ms,0,blend_radius_m)
    movel([0.103808, -1.352274, -2.592164, -0.767951, 1.570796, 1.674604],accel_mss,speed_ms,0,blend_radius_m)
    movel([0.101648, -1.352565, -2.591971, -0.767854, 1.570796, 1.672444],accel_mss,speed_ms,0,blend_radius_m)
    movel([0.100622, -1.352545, -2.591984, -0.767860, 1.570796, 1.671418],accel_mss,speed_ms,0,blend_radius_m)
    movel([0.098747, -1.352187, -2.592222, -0.767980, 1.570796, 1.669544],accel_mss,speed_ms,0,blend_radius_m)
    movel([0.097947, -1.351861, -2.592439, -0.768089, 1.570796, 1.668744],accel_mss,speed_ms,0,blend_radius_m)
    movel([0.096622, -1.350903, -2.593075, -0.768411, 1.570796, 1.667419],accel_mss,speed_ms,0,blend_radius_m)
    movel([0.096111, -1.350283, -2.593486, -0.768620, 1.570796, 1.666907],accel_mss,speed_ms,0,blend_radius_m)
    movel([0.095740, -1.349613, -2.593930, -0.768846, 1.570796, 1.666536],accel_mss,speed_ms,0,blend_radius_m)
    movel([0.095501, -1.348861, -2.594427, -0.769101, 1.570796, 1.666297],accel_mss,speed_ms,0,blend_radius_m)
    movel([0.095395, -1.348037, -2.594971, -0.769381, 1.570796, 1.666191],accel_mss,speed_ms,0,blend_radius_m)
    movel([0.095426, -1.347156, -2.595552, -0.769682, 1.570796, 1.666222],accel_mss,speed_ms,0,blend_radius_m)
    movel([0.095866, -1.345036, -2.596944, -0.770409, 1.570796, 1.666663],accel_mss,speed_ms,0,blend_radius_m)
    movel([0.096222, -1.344064, -2.597580, -0.770745, 1.570796, 1.667018],accel_mss,speed_ms,0,blend_radius_m)
    movel([0.096705, -1.343085, -2.598220, -0.771084, 1.570796, 1.667501],accel_mss,speed_ms,0,blend_radius_m)
    movel([0.097043, -1.342642, -2.598509, -0.771238, 1.570796, 1.667839],accel_mss,speed_ms,0,blend_radius_m)
    movel([0.097498, -1.342288, -2.598740, -0.771361, 1.570796, 1.668295],accel_mss,speed_ms,0,blend_radius_m)
    movel([0.097874, -1.342192, -2.598802, -0.771395, 1.570796, 1.668670],accel_mss,speed_ms,0,blend_radius_m)
    movel([0.098443, -1.342656, -2.598500, -0.771233, 1.570796, 1.669239],accel_mss,speed_ms,0,blend_radius_m)
    movel([0.098748, -1.342710, -2.598464, -0.771214, 1.570796, 1.669544],accel_mss,speed_ms,0,blend_radius_m)
    movel([0.099687, -1.342645, -2.598507, -0.771237, 1.570796, 1.670484],accel_mss,speed_ms,0,blend_radius_m)
    movel([0.100230, -1.342728, -2.598453, -0.771208, 1.570796, 1.671026],accel_mss,speed_ms,0,blend_radius_m)
    movel([0.101769, -1.343304, -2.598077, -0.771008, 1.570796, 1.672565],accel_mss,speed_ms,0,blend_radius_m)
    movel([0.103166, -1.344105, -2.597554, -0.770731, 1.570796, 1.673962],accel_mss,speed_ms,0,blend_radius_m)
    movel([0.103885, -1.344929, -2.597014, -0.770446, 1.570796, 1.674681],accel_mss,speed_ms,0,blend_radius_m)
    movel([0.104469, -1.345525, -2.596623, -0.770241, 1.570796, 1.675266],accel_mss,speed_ms,0,blend_radius_m)
    movel([0.104853, -1.345643, -2.596546, -0.770200, 1.570796, 1.675649],accel_mss,speed_ms,0,blend_radius_m)
    movel([0.105311, -1.345628, -2.596556, -0.770205, 1.570796, 1.676107],accel_mss,speed_ms,0,blend_radius_m)
    movel([0.105774, -1.345486, -2.596649, -0.770254, 1.570796, 1.676570],accel_mss,speed_ms,0,blend_radius_m)
    movel([0.106227, -1.345218, -2.596824, -0.770346, 1.570796, 1.677023],accel_mss,speed_ms,0,blend_radius_m)
    movel([0.107036, -1.344392, -2.597366, -0.770631, 1.570796, 1.677832],accel_mss,speed_ms,0,blend_radius_m)
    movel([0.107279, -1.343954, -2.597652, -0.770783, 1.570796, 1.678075],accel_mss,speed_ms,0,blend_radius_m)
    movel([0.107400, -1.343518, -2.597937, -0.770934, 1.570796, 1.678197],accel_mss,speed_ms,0,blend_radius_m)
    movel([0.107388, -1.343128, -2.598192, -0.771069, 1.570796, 1.678184],accel_mss,speed_ms,0,blend_radius_m)
    movel([0.106943, -1.342535, -2.598579, -0.771275, 1.570796, 1.677739],accel_mss,speed_ms,0,blend_radius_m)
    movel([0.106546, -1.342368, -2.598688, -0.771333, 1.570796, 1.677343],accel_mss,speed_ms,0,blend_radius_m)
    movel([0.104127, -1.342161, -2.598823, -0.771406, 1.570796, 1.674923],accel_mss,speed_ms,0,blend_radius_m)
    movel([0.102587, -1.341632, -2.599167, -0.771590, 1.570796, 1.673384],accel_mss,speed_ms,0,blend_radius_m)
    movel([0.101253, -1.340948, -2.599611, -0.771829, 1.570796, 1.672050],accel_mss,speed_ms,0,blend_radius_m)
    movel([0.101043, -1.340707, -2.599768, -0.771914, 1.570796, 1.671839],accel_mss,speed_ms,0,blend_radius_m)
    movel([0.100948, -1.340168, -2.600118, -0.772103, 1.570796, 1.671745],accel_mss,speed_ms,0,blend_radius_m)
    movel([0.100740, -1.340015, -2.600217, -0.772157, 1.570796, 1.671536],accel_mss,speed_ms,0,blend_radius_m)
    movel([0.099656, -1.339836, -2.600333, -0.772220, 1.570796, 1.670452],accel_mss,speed_ms,0,blend_radius_m)
    movel([0.100127, -1.339181, -2.600758, -0.772450, 1.570796, 1.670924],accel_mss,speed_ms,0,blend_radius_m)
    movel([0.101463, -1.338205, -2.601389, -0.772795, 1.570796, 1.672259],accel_mss,speed_ms,0,blend_radius_m)
    movel([0.102861, -1.337276, -2.601988, -0.773125, 1.570796, 1.673658],accel_mss,speed_ms,0,blend_radius_m)
    movel([0.104075, -1.336636, -2.602401, -0.773352, 1.570796, 1.674871],accel_mss,speed_ms,0,blend_radius_m)
    movel([0.105399, -1.336140, -2.602720, -0.773529, 1.570796, 1.676196],accel_mss,speed_ms,0,blend_radius_m)
    movel([0.107177, -1.335653, -2.603033, -0.773703, 1.570796, 1.677973],accel_mss,speed_ms,0,blend_radius_m)
    movel([0.108601, -1.335371, -2.603214, -0.773804, 1.570796, 1.679398],accel_mss,speed_ms,0,blend_radius_m)
    movel([0.109986, -1.335226, -2.603307, -0.773856, 1.570796, 1.680782],accel_mss,speed_ms,0,blend_radius_m)
    movel([0.111169, -1.335247, -2.603294, -0.773849, 1.570796, 1.681965],accel_mss,speed_ms,0,blend_radius_m)
    movel([0.112261, -1.335436, -2.603172, -0.773781, 1.570796, 1.683057],accel_mss,speed_ms,0,blend_radius_m)
    movel([0.113195, -1.335783, -2.602949, -0.773657, 1.570796, 1.683991],accel_mss,speed_ms,0,blend_radius_m)
    movel([0.113992, -1.336289, -2.602624, -0.773476, 1.570796, 1.684789],accel_mss,speed_ms,0,blend_radius_m)
    movel([0.114668, -1.336964, -2.602189, -0.773236, 1.570796, 1.685464],accel_mss,speed_ms,0,blend_radius_m)
    movel([0.115189, -1.337765, -2.601673, -0.772951, 1.570796, 1.685985],accel_mss,speed_ms,0,blend_radius_m)
    movel([0.115742, -1.339291, -2.600686, -0.772412, 1.570796, 1.686539],accel_mss,speed_ms,0,blend_radius_m)
    movel([0.115839, -1.340013, -2.600218, -0.772157, 1.570796, 1.686635],accel_mss,speed_ms,0,blend_radius_m)
    movel([0.115658, -1.341596, -2.599190, -0.771603, 1.570796, 1.686454],accel_mss,speed_ms,0,blend_radius_m)
    movel([0.115384, -1.342429, -2.598648, -0.771312, 1.570796, 1.686180],accel_mss,speed_ms,0,blend_radius_m)
    movel([0.114436, -1.344399, -2.597361, -0.770629, 1.570796, 1.685232],accel_mss,speed_ms,0,blend_radius_m)
    movel([0.113833, -1.345365, -2.596728, -0.770296, 1.570796, 1.684629],accel_mss,speed_ms,0,blend_radius_m)
    movel([0.113126, -1.346300, -2.596115, -0.769975, 1.570796, 1.683923],accel_mss,speed_ms,0,blend_radius_m)
    movel([0.112740, -1.346706, -2.595848, -0.769836, 1.570796, 1.683536],accel_mss,speed_ms,0,blend_radius_m)
    speed_ms = 0.005
    movel([0.112740, -1.337761, -2.591699, -0.782928, 1.570796, 1.683536],accel_mss,speed_ms,0,blend_radius_m)
    speed_ms = 0.040
    movel([0.119109, -1.320588, -2.602645, -0.789155, 1.570796, 1.689905],accel_mss,speed_ms,0,blend_radius_m)
    speed_ms = 0.005
    movel([0.119109, -1.329642, -2.606870, -0.775876, 1.570796, 1.689905],accel_mss,speed_ms,0,blend_radius_m)
    speed_ms = 0.030
    movel([0.119398, -1.329751, -2.606802, -0.775837, 1.570796, 1.690195],accel_mss,speed_ms,0,blend_radius_m)
    movel([0.119518, -1.330014, -2.606634, -0.775741, 1.570796, 1.690314],accel_mss,speed_ms,0,blend_radius_m)
    movel([0.119516, -1.331479, -2.605703, -0.775207, 1.570796, 1.690312],accel_mss,speed_ms,0,blend_radius_m)
    movel([0.119225, -1.334201, -2.603965, -0.774224, 1.570796, 1.690022],accel_mss,speed_ms,0,blend_radius_m)
    movel([0.116814, -1.350716, -2.593199, -0.768474, 1.570796, 1.687610],accel_mss,speed_ms,0,blend_radius_m)
    movel([0.104155, -1.354449, -2.590714, -0.767226, 1.570796, 1.674951],accel_mss,speed_ms,0,blend_radius_m)
    movel([0.094111, -1.357371, -2.588754, -0.766263, 1.570796, 1.664908],accel_mss,speed_ms,0,blend_radius_m)
    movel([0.091721, -1.357962, -2.588357, -0.766070, 1.570796, 1.662517],accel_mss,speed_ms,0,blend_radius_m)
    movel([0.091406, -1.357967, -2.588354, -0.766068, 1.570796, 1.662202],accel_mss,speed_ms,0,blend_radius_m)
    movel([0.091183, -1.357835, -2.588443, -0.766112, 1.570796, 1.661979],accel_mss,speed_ms,0,blend_radius_m)
    movel([0.090901, -1.357259, -2.588830, -0.766300, 1.570796, 1.661698],accel_mss,speed_ms,0,blend_radius_m)
    movel([0.090858, -1.356557, -2.589301, -0.766530, 1.570796, 1.661654],accel_mss,speed_ms,0,blend_radius_m)
    movel([0.091818, -1.347808, -2.595122, -0.769459, 1.570796, 1.662615],accel_mss,speed_ms,0,blend_radius_m)
    movel([0.092892, -1.338787, -2.601013, -0.772590, 1.570796, 1.663688],accel_mss,speed_ms,0,blend_radius_m)
    movel([0.093093, -1.338166, -2.601414, -0.772809, 1.570796, 1.663890],accel_mss,speed_ms,0,blend_radius_m)
    movel([0.093526, -1.337557, -2.601807, -0.773025, 1.570796, 1.664322],accel_mss,speed_ms,0,blend_radius_m)
    movel([0.094082, -1.337087, -2.602110, -0.773192, 1.570796, 1.664878],accel_mss,speed_ms,0,blend_radius_m)
    movel([0.094712, -1.336784, -2.602305, -0.773300, 1.570796, 1.665509],accel_mss,speed_ms,0,blend_radius_m)
    movel([0.116851, -1.329939, -2.606682, -0.775768, 1.570796, 1.687647],accel_mss,speed_ms,0,blend_radius_m)
    movel([0.118012, -1.329690, -2.606840, -0.775859, 1.570796, 1.688809],accel_mss,speed_ms,0,blend_radius_m)
    movel([0.119109, -1.329642, -2.606870, -0.775876, 1.570796, 1.689905],accel_mss,speed_ms,0,blend_radius_m)
    movel([0.119398, -1.329751, -2.606802, -0.775837, 1.570796, 1.690195],accel_mss,speed_ms,0,blend_radius_m)
    movel([0.119518, -1.330014, -2.606634, -0.775741, 1.570796, 1.690314],accel_mss,speed_ms,0,blend_radius_m)
    movel([0.119516, -1.331479, -2.605703, -0.775207, 1.570796, 1.690312],accel_mss,speed_ms,0,blend_radius_m)
    speed_ms = 0.005
    movel([0.119503, -1.322565, -2.601406, -0.788419, 1.570796, 1.690300],accel_mss,speed_ms,0,blend_radius_m)
    speed_ms = 0.040
    movel([0.113728, -1.303865, -2.612930, -0.795595, 1.570796, 1.684524],accel_mss,speed_ms,0,blend_radius_m)
    speed_ms = 0.005
    movel([0.113728, -1.313020, -2.617229, -0.782139, 1.570796, 1.684524],accel_mss,speed_ms,0,blend_radius_m)
    speed_ms = 0.030
    movel([0.092754, -1.319668, -2.613131, -0.779590, 1.570796, 1.663550],accel_mss,speed_ms,0,blend_radius_m)
    movel([0.095175, -1.297035, -2.626848, -0.788506, 1.570796, 1.665971],accel_mss,speed_ms,0,blend_radius_m)
    movel([0.097729, -1.273585, -2.640364, -0.798440, 1.570796, 1.668525],accel_mss,speed_ms,0,blend_radius_m)
    movel([0.120006, -1.266167, -2.644496, -0.801726, 1.570796, 1.690802],accel_mss,speed_ms,0,blend_radius_m)
    movel([0.142413, -1.259043, -2.648400, -0.804946, 1.570796, 1.713209],accel_mss,speed_ms,0,blend_radius_m)
    movel([0.138512, -1.283289, -2.634855, -0.794245, 1.570796, 1.709308],accel_mss,speed_ms,0,blend_radius_m)
    movel([0.134816, -1.306640, -2.621108, -0.784640, 1.570796, 1.705613],accel_mss,speed_ms,0,blend_radius_m)
    movel([0.113728, -1.313020, -2.617229, -0.782139, 1.570796, 1.684524],accel_mss,speed_ms,0,blend_radius_m)
    movel([0.111014, -1.313864, -2.616712, -0.781812, 1.570796, 1.681811],accel_mss,speed_ms,0,blend_radius_m)
    speed_ms = 0.005
    movel([0.111014, -1.304713, -2.612417, -0.795259, 1.570796, 1.681811],accel_mss,speed_ms,0,blend_radius_m)
    speed_ms = 0.040
    movel([0.082365, -1.325148, -2.599778, -0.787463, 1.570796, 1.653161],accel_mss,speed_ms,0,blend_radius_m)
    speed_ms = 0.005
    movel([0.082365, -1.334173, -2.603982, -0.774234, 1.570796, 1.653161],accel_mss,speed_ms,0,blend_radius_m)
    speed_ms = 0.030
    movel([0.076943, -1.335786, -2.602947, -0.773656, 1.570796, 1.647739],accel_mss,speed_ms,0,blend_radius_m)
    movel([0.077382, -1.329257, -2.607114, -0.776017, 1.570796, 1.648179],accel_mss,speed_ms,0,blend_radius_m)
    movel([0.077826, -1.322665, -2.611264, -0.778460, 1.570796, 1.648622],accel_mss,speed_ms,0,blend_radius_m)
    movel([0.083497, -1.320809, -2.612421, -0.779159, 1.570796, 1.654293],accel_mss,speed_ms,0,blend_radius_m)
    movel([0.089175, -1.318972, -2.613562, -0.779854, 1.570796, 1.659971],accel_mss,speed_ms,0,blend_radius_m)
    movel([0.088479, -1.325811, -2.609291, -0.777287, 1.570796, 1.659275],accel_mss,speed_ms,0,blend_radius_m)
    movel([0.087793, -1.332579, -2.605001, -0.774808, 1.570796, 1.658590],accel_mss,speed_ms,0,blend_radius_m)
    movel([0.082365, -1.334173, -2.603982, -0.774234, 1.570796, 1.653161],accel_mss,speed_ms,0,blend_radius_m)
    movel([0.079719, -1.334957, -2.603479, -0.773952, 1.570796, 1.650515],accel_mss,speed_ms,0,blend_radius_m)
    speed_ms = 0.005
    movel([0.079719, -1.325937, -2.599279, -0.787173, 1.570796, 1.650515],accel_mss,speed_ms,0,blend_radius_m)
    speed_ms = 0.040
    movel([0.069921, -1.329195, -2.597209, -0.785985, 1.570796, 1.640717],accel_mss,speed_ms,0,blend_radius_m)
    speed_ms = 0.005
    movel([0.069921, -1.338195, -2.601395, -0.772799, 1.570796, 1.640717],accel_mss,speed_ms,0,blend_radius_m)
    speed_ms = 0.030
    movel([0.064499, -1.340106, -2.600158, -0.772125, 1.570796, 1.635295],accel_mss,speed_ms,0,blend_radius_m)
    movel([0.064998, -1.333471, -2.604431, -0.774486, 1.570796, 1.635794],accel_mss,speed_ms,0,blend_radius_m)
    movel([0.065505, -1.326770, -2.608686, -0.776932, 1.570796, 1.636301],accel_mss,speed_ms,0,blend_radius_m)
    movel([0.070780, -1.325000, -2.609800, -0.777588, 1.570796, 1.641576],accel_mss,speed_ms,0,blend_radius_m)
    movel([0.074610, -1.323820, -2.610541, -0.778028, 1.570796, 1.645406],accel_mss,speed_ms,0,blend_radius_m)
    movel([0.076099, -1.323423, -2.610790, -0.778177, 1.570796, 1.646895],accel_mss,speed_ms,0,blend_radius_m)
    movel([0.076407, -1.323448, -2.610774, -0.778167, 1.570796, 1.647203],accel_mss,speed_ms,0,blend_radius_m)
    movel([0.076527, -1.323690, -2.610622, -0.778077, 1.570796, 1.647323],accel_mss,speed_ms,0,blend_radius_m)
    movel([0.076292, -1.327562, -2.608187, -0.776640, 1.570796, 1.647089],accel_mss,speed_ms,0,blend_radius_m)
    movel([0.076046, -1.330006, -2.606640, -0.775744, 1.570796, 1.646843],accel_mss,speed_ms,0,blend_radius_m)
    movel([0.075354, -1.336299, -2.602617, -0.773472, 1.570796, 1.646150],accel_mss,speed_ms,0,blend_radius_m)
    movel([0.069921, -1.338195, -2.601395, -0.772799, 1.570796, 1.640717],accel_mss,speed_ms,0,blend_radius_m)
    movel([0.067274, -1.339126, -2.600793, -0.772470, 1.570796, 1.638071],accel_mss,speed_ms,0,blend_radius_m)
    speed_ms = 0.005
    movel([0.067274, -1.330132, -2.596611, -0.785646, 1.570796, 1.638071],accel_mss,speed_ms,0,blend_radius_m)
    speed_ms = 0.040
    movel([0.075000, -1.343145, -2.588186, -0.781058, 1.570796, 1.645797],accel_mss,speed_ms,0,blend_radius_m)
    speed_ms = 0.005
    movel([0.075000, -1.352054, -2.592310, -0.768024, 1.570796, 1.645797],accel_mss,speed_ms,0,blend_radius_m)
    speed_ms = 0.030
    movel([0.062813, -1.355951, -2.589708, -0.766730, 1.570796, 1.633609],accel_mss,speed_ms,0,blend_radius_m)
    movel([0.063322, -1.349042, -2.594307, -0.769039, 1.570796, 1.634118],accel_mss,speed_ms,0,blend_radius_m)
    movel([0.063839, -1.342062, -2.598887, -0.771440, 1.570796, 1.634635],accel_mss,speed_ms,0,blend_radius_m)
    movel([0.076231, -1.338019, -2.601509, -0.772861, 1.570796, 1.647027],accel_mss,speed_ms,0,blend_radius_m)
    movel([0.088671, -1.334064, -2.604052, -0.774273, 1.570796, 1.659467],accel_mss,speed_ms,0,blend_radius_m)
    movel([0.087946, -1.341192, -2.599453, -0.771744, 1.570796, 1.658742],accel_mss,speed_ms,0,blend_radius_m)
    movel([0.087233, -1.348244, -2.594835, -0.769311, 1.570796, 1.658029],accel_mss,speed_ms,0,blend_radius_m)
    movel([0.075000, -1.352054, -2.592310, -0.768024, 1.570796, 1.645797],accel_mss,speed_ms,0,blend_radius_m)
    movel([0.072403, -1.352876, -2.591763, -0.767750, 1.570796, 1.643200],accel_mss,speed_ms,0,blend_radius_m)
    speed_ms = 0.005
    movel([0.072403, -1.343972, -2.587642, -0.780774, 1.570796, 1.643200],accel_mss,speed_ms,0,blend_radius_m)
    speed_ms = 0.040
    movel([0.074469, -1.346376, -2.586058, -0.779955, 1.570796, 1.645266],accel_mss,speed_ms,0,blend_radius_m)
    speed_ms = 0.005
    movel([0.074469, -1.355264, -2.590168, -0.766956, 1.570796, 1.645266],accel_mss,speed_ms,0,blend_radius_m)
    speed_ms = 0.030
    movel([0.081798, -1.352961, -2.591707, -0.767721, 1.570796, 1.652595],accel_mss,speed_ms,0,blend_radius_m)
    movel([0.084331, -1.352077, -2.592295, -0.768017, 1.570796, 1.655127],accel_mss,speed_ms,0,blend_radius_m)
    movel([0.085519, -1.351463, -2.592704, -0.768223, 1.570796, 1.656315],accel_mss,speed_ms,0,blend_radius_m)
    movel([0.085828, -1.351165, -2.592901, -0.768323, 1.570796, 1.656625],accel_mss,speed_ms,0,blend_radius_m)
    movel([0.085966, -1.350821, -2.593129, -0.768438, 1.570796, 1.656762],accel_mss,speed_ms,0,blend_radius_m)
    movel([0.085890, -1.350543, -2.593314, -0.768532, 1.570796, 1.656686],accel_mss,speed_ms,0,blend_radius_m)
    movel([0.085622, -1.350422, -2.593394, -0.768573, 1.570796, 1.656418],accel_mss,speed_ms,0,blend_radius_m)
    movel([0.084482, -1.350524, -2.593326, -0.768538, 1.570796, 1.655279],accel_mss,speed_ms,0,blend_radius_m)
    movel([0.081965, -1.351200, -2.592878, -0.768311, 1.570796, 1.652762],accel_mss,speed_ms,0,blend_radius_m)
    movel([0.074624, -1.353479, -2.591362, -0.767549, 1.570796, 1.645420],accel_mss,speed_ms,0,blend_radius_m)
    movel([0.067296, -1.355824, -2.589794, -0.766772, 1.570796, 1.638093],accel_mss,speed_ms,0,blend_radius_m)
    movel([0.064774, -1.356735, -2.589182, -0.766472, 1.570796, 1.635570],accel_mss,speed_ms,0,blend_radius_m)
    movel([0.063597, -1.357360, -2.588762, -0.766267, 1.570796, 1.634394],accel_mss,speed_ms,0,blend_radius_m)
    movel([0.063295, -1.357658, -2.588561, -0.766169, 1.570796, 1.634092],accel_mss,speed_ms,0,blend_radius_m)
    movel([0.063167, -1.357998, -2.588333, -0.766058, 1.570796, 1.633963],accel_mss,speed_ms,0,blend_radius_m)
    movel([0.063250, -1.358269, -2.588150, -0.765970, 1.570796, 1.634047],accel_mss,speed_ms,0,blend_radius_m)
    movel([0.063521, -1.358382, -2.588074, -0.765933, 1.570796, 1.634318],accel_mss,speed_ms,0,blend_radius_m)
    movel([0.064659, -1.358262, -2.588155, -0.765972, 1.570796, 1.635455],accel_mss,speed_ms,0,blend_radius_m)
    movel([0.067160, -1.357563, -2.588626, -0.766201, 1.570796, 1.637956],accel_mss,speed_ms,0,blend_radius_m)
    movel([0.074469, -1.355264, -2.590168, -0.766956, 1.570796, 1.645266],accel_mss,speed_ms,0,blend_radius_m)
    movel([0.077059, -1.354446, -2.590716, -0.767227, 1.570796, 1.647855],accel_mss,speed_ms,0,blend_radius_m)
    speed_ms = 0.005
    movel([0.077059, -1.345552, -2.586602, -0.780235, 1.570796, 1.647855],accel_mss,speed_ms,0,blend_radius_m)
    speed_ms = 0.040
    movel([0.074315, -1.348169, -2.584872, -0.779349, 1.570796, 1.645111],accel_mss,speed_ms,0,blend_radius_m)
    speed_ms = 0.005
    movel([0.074315, -1.357045, -2.588974, -0.766370, 1.570796, 1.645111],accel_mss,speed_ms,0,blend_radius_m)
    speed_ms = 0.030
    movel([0.065941, -1.359582, -2.587264, -0.765543, 1.570796, 1.636738],accel_mss,speed_ms,0,blend_radius_m)
    movel([0.063213, -1.360336, -2.586755, -0.765299, 1.570796, 1.634009],accel_mss,speed_ms,0,blend_radius_m)
    movel([0.063004, -1.360205, -2.586843, -0.765341, 1.570796, 1.633800],accel_mss,speed_ms,0,blend_radius_m)
    movel([0.063243, -1.359930, -2.587029, -0.765430, 1.570796, 1.634039],accel_mss,speed_ms,0,blend_radius_m)
    movel([0.069538, -1.357713, -2.588525, -0.766151, 1.570796, 1.640335],accel_mss,speed_ms,0,blend_radius_m)
    movel([0.074392, -1.356155, -2.589571, -0.766663, 1.570796, 1.645188],accel_mss,speed_ms,0,blend_radius_m)
    movel([0.082794, -1.353654, -2.591245, -0.767490, 1.570796, 1.653590],accel_mss,speed_ms,0,blend_radius_m)
    movel([0.085537, -1.352933, -2.591726, -0.767731, 1.570796, 1.656334],accel_mss,speed_ms,0,blend_radius_m)
    movel([0.085742, -1.353070, -2.591634, -0.767685, 1.570796, 1.656539],accel_mss,speed_ms,0,blend_radius_m)
    movel([0.085496, -1.353346, -2.591450, -0.767593, 1.570796, 1.656293],accel_mss,speed_ms,0,blend_radius_m)
    movel([0.079171, -1.355504, -2.590008, -0.766877, 1.570796, 1.649968],accel_mss,speed_ms,0,blend_radius_m)
    movel([0.074315, -1.357045, -2.588974, -0.766370, 1.570796, 1.645111],accel_mss,speed_ms,0,blend_radius_m)
    movel([0.071737, -1.357821, -2.588452, -0.766116, 1.570796, 1.642533],accel_mss,speed_ms,0,blend_radius_m)
    speed_ms = 0.005
    movel([0.071737, -1.348950, -2.584353, -0.779086, 1.570796, 1.642533],accel_mss,speed_ms,0,blend_radius_m)
    speed_ms = 0.040
    movel([0.074162, -1.349957, -2.583684, -0.778748, 1.570796, 1.644958],accel_mss,speed_ms,0,blend_radius_m)
    speed_ms = 0.005
    movel([0.074162, -1.358821, -2.587778, -0.765790, 1.570796, 1.644958],accel_mss,speed_ms,0,blend_radius_m)
    speed_ms = 0.030
    movel([0.079007, -1.357287, -2.588811, -0.766291, 1.570796, 1.649804],accel_mss,speed_ms,0,blend_radius_m)
    movel([0.085319, -1.355139, -2.590252, -0.766998, 1.570796, 1.656115],accel_mss,speed_ms,0,blend_radius_m)
    movel([0.085564, -1.354864, -2.590436, -0.767089, 1.570796, 1.656361],accel_mss,speed_ms,0,blend_radius_m)
    movel([0.085360, -1.354727, -2.590528, -0.767134, 1.570796, 1.656156],accel_mss,speed_ms,0,blend_radius_m)
    movel([0.082622, -1.355444, -2.590048, -0.766897, 1.570796, 1.653419],accel_mss,speed_ms,0,blend_radius_m)
    movel([0.074238, -1.357933, -2.588376, -0.766079, 1.570796, 1.645035],accel_mss,speed_ms,0,blend_radius_m)
    movel([0.069395, -1.359484, -2.587330, -0.765574, 1.570796, 1.640191],accel_mss,speed_ms,0,blend_radius_m)
    movel([0.063113, -1.361691, -2.585836, -0.764861, 1.570796, 1.633909],accel_mss,speed_ms,0,blend_radius_m)
    movel([0.062874, -1.361965, -2.585650, -0.764773, 1.570796, 1.633671],accel_mss,speed_ms,0,blend_radius_m)
    movel([0.063083, -1.362096, -2.585562, -0.764732, 1.570796, 1.633879],accel_mss,speed_ms,0,blend_radius_m)
    movel([0.065805, -1.361346, -2.586070, -0.764972, 1.570796, 1.636602],accel_mss,speed_ms,0,blend_radius_m)
    movel([0.074162, -1.358821, -2.587778, -0.765790, 1.570796, 1.644958],accel_mss,speed_ms,0,blend_radius_m)
    movel([0.076741, -1.358003, -2.588329, -0.766056, 1.570796, 1.647537],accel_mss,speed_ms,0,blend_radius_m)
    speed_ms = 0.005
    movel([0.076741, -1.315346, -2.567258, -0.829785, 1.570796, 1.647537],accel_mss,speed_ms,0,blend_radius_m)
    speed_ms = 1.000
    movel([0.076741, -1.226320, -2.508842, -0.977226, 1.570796, 1.647537],accel_mss,speed_ms,0,blend_radius_m)
    # End of main program
  end

  Machining3()
end
